Fanuc KAREL source: TRANSLATE.kl

PROGRAM T
%NOLOCKGROUP
VAR
 v0 : STRING[40]
 v1 : BOOLEAN
 v2 : INTEGER
BEGIN
 TRANSLATE(v0, v1, v2)
END T
